GLOBALCONSTANTS Modules_with_low_IO_density (* Global constants *)
  (* Standard: 61499-1 *)
  (* Version 1.0, 2024-01-25, franz *)
  VAR_GLOBAL CONSTANT
    LO_00 : USINT := 217;
    LO_01 : USINT := 218;
    LO_02 : USINT := 219;
    LO_03 : USINT := 220;
    LO_04 : USINT := 221;
    LO_05 : USINT := 222;
    LO_06 : USINT := 223;
    LO_07 : USINT := 224;
  END_VAR
END_GLOBALCONSTANTS
